FUNCTION Call_Remover

instRemoverConveyorOutfeedLong(PartPresent:= SensorConveyorOutfeedEnd, 
					   	  	   ActorInstanceIndex := 0,
					   	  	   ActorInstanceName := 'FeedOut',
					   	  	   HMIInterface := hmiMachineSectionInterface,
						  	   OperatingModeSection := instOperatingMode.StateOperatingMode,
					   	  	   RemovePart=> ConveyorFeedOutLongRemover);

instRemoverConveyorOutfeedLong.Remove();

END_FUNCTION

(* stored: Version 1.1.0.1
   POU Call_Remover: Id {4486a922-5b20-46e7-8b7f-272c76e02a85}, SpecialFunc None *)
